(* PLC project seal_in, plcc plcc tests 1 *)
(* stored: creationDateTime 2026-09-27T00:00:00 *)

PROGRAM SealIn
  VAR
    Start AT %IX0.0 : BOOL;
    Stop AT %IX0.1 : BOOL;
    Motor AT %QX0.0 : BOOL;
  END_VAR

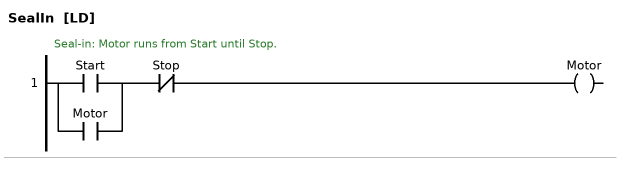
(* LD diagram, written out as Structured Text *)
(* Seal-in: Motor runs from Start until Stop. *)
Motor := (Start OR Motor) AND NOT Stop;
END_PROGRAM

CONFIGURATION Config0
  RESOURCE Res0 ON PLC
    TASK MainTask(INTERVAL := T#20ms, PRIORITY := 0);
    PROGRAM seal WITH MainTask : SealIn;
  END_RESOURCE
END_CONFIGURATION
